// TIA Portal V19 export
TYPE "Valve"
   STRUCT
      ManOpen : Bool;
      FeebackFitted : Bool;
      ValveisOpen : Bool;
      ValveisClosed : Bool;
      ValveAngle : Real;
      FeedbackFaultTime : Time;
   END_STRUCT;
END_TYPE
